TYPE EL3443_Phase_Basic :
STRUCT
END_STRUCT
END_TYPE

(* stored: Version 1.1.0.1, ProductVersion 3.1.4024.12
   DUT EL3443_Phase_Basic: Id {a8e6e8ac-3b79-4e29-8e9c-81592f10909e} *)
